TYPE csp_transfer_main_brand_case_pattern :
STRUCT
	
	case_pattern_L:								INT := 2; (*$P min := 0; max := 5; step := 1; unit := u ; desc := Case Pattern L; $*)
	case_pattern_W:								INT := 2; (*$P min := 0; max := 5; step := 1; unit := u; desc := Case Pattern W; $*)
	case_pattern_D:								INT := 1; (*$P min := 0; max := 5; step := 1; unit := u; desc := Case Pattern D; $*)
			
END_STRUCT
END_TYPE

(* stored: Version 1.1.0.1, ProductVersion 3.1.4024.3
   DUT csp_transfer_main_brand_case_pattern: Id {e2818816-d98a-45ee-987d-9b57947afb8b} *)
